PROGRAM P_Demo_FB_JsonDomParser_LoadDocumentFromFile
VAR
    fbParser : FB_JsonDomParser; // 父 FB 实例
    bExecRaw : BOOL; // 给 bExec 用的具名后备变量
    sFile : STRING(255);
    hrErrorCode : HRESULT;
    vRet : BOOL; // 返回值监视
    bTrigger : BOOL := FALSE; // 在线置 TRUE 触发一次调用
    bTriggerPrev : BOOL;
END_VAR

// =============================================================================
// 场景：PLC 启动时从 SD 卡里读一份缓存的配方 JSON，无需上位机推送。
// 价值：一次调用完成异步读盘 + UTF-8 解码 + DOM 解析，无需自己写文件 IO 链。
// 验证：登录 PLC 在线写 bTrigger := TRUE 触发，monitor 返回值/输出参数。具体步骤见下方注释。
// 验证步骤：
//   1. 右键 PLC 项目下 POUs 文件夹 → Add → Existing Item → 选本 .TcPOU 文件
//   2. 引用 Tc3_JsonXml（References → Add library）
//   3. 编译 → 登录 → 运行；按 verify 注释里给出的在线写值操作
// =============================================================================

// 上升沿触发一次方法调用并观察输出。
IF bTrigger AND NOT bTriggerPrev THEN
    vRet := fbParser.LoadDocumentFromFile(
        bExec := bExecRaw,
        sFile := sFile,
        hrErrorCode => hrErrorCode
    );
END_IF;
bTriggerPrev := bTrigger;

END_PROGRAM

(* stored: Version 1.1.0.1, ProductVersion 3.1.4024.5
   POU P_Demo_FB_JsonDomParser_LoadDocumentFromFile: Id {6f88bcb6-d666-5aed-b4b8-072ce2ec1e4f}, SpecialFunc None *)
